TYPE ST_Complex :
STRUCT
	bMember 		: BOOL;
	eMember 		: E_Enum;
	stSimpleMember 	: ST_Simple;
    stPackedMember 	: ST_Packed;
	fbMember 		: FB_Simple(TRUE, 99, 'Complex Test.');
	arrfMember 		: ARRAY[0..2] OF LREAL;
END_STRUCT
END_TYPE

(* stored: Version 1.1.0.1
   DUT ST_Complex: Id {68321886-0b96-4052-9841-5a582aafe8a4} *)
